{attribute 'linkalways'} 
{attribute 'no_explicit_call' := 'This FB is a CLASS and must be accessed using methods or properties'}
{attribute 'enable_dynamic_creation'}
FUNCTION_BLOCK ABSTRACT CollectionEvent EXTENDS Disposable
VAR
	_target : I_Collection;
END_VAR

METHOD FB_init : BOOL
VAR_INPUT
	bInitRetains : BOOL; // if TRUE, the retain variables are initialized (warm start / cold start)
	bInCopyCode : BOOL;  // if TRUE, the instance afterwards gets moved into the copy code (online change)
	Target : I_Collection;
END_VAR
This^._target := Target;
END_METHOD

PROPERTY PUBLIC Target : I_Collection
GET // PUBLIC
Target := _target;
END_GET
END_PROPERTY

END_FUNCTION_BLOCK

(* stored: Version 1.1.0.1, ProductVersion 3.1.4024.12
   POU CollectionEvent: Id {b0c7c138-9fb1-01b9-3330-8121a5f03fd9}, SpecialFunc None
   Folder Constructor: Id {ace252f8-71f4-0d0b-22be-57613ae1b5d9}
   Method FB_init: Id {4cef3445-a1aa-0a7a-1b27-e87e47d04019}
   Property Target: Id {5d8f4459-a1c9-03b8-1617-258433dddfea}
   Get Get: Id {8195f2de-9ab4-0158-33bf-f455378fc2ee} *)
